PROGRAM PLC_TASK_1
VAR
END_VAR

PRG_PowerSlits();

END_PROGRAM

(* stored: Version 1.1.0.1, ProductVersion 3.1.4022.18
   POU PLC_TASK_1: Id {d99ae9cd-8a5b-44cf-9736-9f9943eefa8f}, SpecialFunc None *)
